TYPE EL1xx9_Data :
STRUCT
	{attribute addProperty Name "1"}
	{attribute addProperty Name "Channel 1"}
	_1 :DiChannel;
	{attribute addProperty Name "Channel 2"}
	_2 :DiChannel;
	{attribute addProperty Name "Channel 3"}
	_3 :DiChannel;
	{attribute addProperty Name "Channel 4"}
	_4 :DiChannel;
	{attribute addProperty Name "Channel 5"}
	_5 :DiChannel;
	{attribute addProperty Name "Channel 6"}
	_6 :DiChannel;
	{attribute addProperty Name "Channel 7"}
	_7 :DiChannel;
	{attribute addProperty Name "Channel 8"}
	_8 :DiChannel;
	{attribute addProperty Name "Channel 9"}
	_9 :DiChannel;
	{attribute addProperty Name "Channel 10"}
	_10 :DiChannel;
	{attribute addProperty Name "Channel 11"}
	_11 :DiChannel;
	{attribute addProperty Name "Channel 12"}
	_12 :DiChannel;
	{attribute addProperty Name "Channel 13"}
	_13 :DiChannel;
	{attribute addProperty Name "Channel 14"}
	_14 :DiChannel;
	{attribute addProperty Name "Channel 15"}
	_15 :DiChannel;
	{attribute addProperty Name "Channel 16"}
	_16 :DiChannel;
END_STRUCT
END_TYPE

(* stored: Version 1.1.0.1, ProductVersion 3.1.4024.9
   DUT EL1xx9_Data: Id {29d01bfb-4e9b-0710-1c40-9588df811326} *)
